{attribute 'GeneratedUsingTerminal: EK1100-0000-0018'}
{attribute addProperty BoxType "EK1100-0000-0018"}
{attribute addProperty Id "Beckhoff_EL72xxEK1122Beckhoff_EL72xxEK1122_48DD6FE82A_0001_EL7201_0000_0017EL7201_E258D19D33A_0002_EL7201_0000_0018EL7201_E258D19D33A_0003_EL7201_0000_0019EL7201_E258D19D33A_0004_EL7201_0000_0020EL7201_E258D19D33A_0005_EL7201_0000_0021EL7201_E258D19D33A_0006_EL7201_0001_0017EL7201_2B9C00AB33A_0007_EL7201_0001_0018EL7201_2B9C00AB33A_0008_EL7201_0001_0019EL7201_2B9C00AB33A_0009_EL7201_0001_0020EL7201_2B9C00AB33A_0010_EL7201_0001_0021EL7201_2B9C00AB33A_0011_EL7201_0010_0019EL7201_E258D19D33A_0012_EL7201_0010_0020EL7201_E258D19D33A_0013_EL7201_0010_0021EL7201_E258D19D33A_0014_EL7201_0010_0022EL7201_E258D19D33A_0015_EL7201_0010_0023EL7201_E258D19D33A_0016_EL7201_0010_0024EL7201_E258D19D33A_0017_EL7201_0010_0025EL7201_E258D19D33A_0018_EL7201_0010_0026EL7201_E258D19D33A_0019_EL7201_0010_0027EL7201_E258D19D33A_0020_EL7201_0010_0028EL7201_E258D19D33A_0021_EL7201_0010_0029EL7201_E258D19D33A_0022_EL7201_0010_0030EL7201_D07AE8BA34A_0023_EL7201_0010_0031EL7201_D07AE8BA34A_0024_EL7201_0010_0032EL7201_D07AE8BA34A_0025_EL7201_0011_0019EL7201_2B9C00AB33A_0026_EL7201_0011_0020EL7201_2B9C00AB33A_0027_EL7201_0011_0021EL7201_2B9C00AB33A_0028_EL7201_0011_0022EL7201_2B9C00AB33A_0029_EL7201_0011_0023EL7201_2B9C00AB33A_0030_EL7201_0011_0024EL7201_2B9C00AB33A_0031_EL7201_0011_0025EL7201_2B9C00AB33A_0032_EL7201_0011_0026EL7201_2B9C00AB33A_0033_EL7201_0011_0027EL7201_2B9C00AB33A_0034_EL7201_0011_0028EL7201_2B9C00AB33A_0035_EL7201_0011_0029EL7201_2B9C00AB33A_0036_EL7201_0011_0030EL7201_2B9C00AB33A_0037_EL7201_0011_0031EL7201_2B9C00AB33A_0038_EL7201_0011_0032EL7201_2B9C00AB33A_0039_EL7211_0000_0020EL7211_E258D19D33A_0040_EL7211_0000_0021EL7211_E258D19D33A_0041_EL7211_0001_0020EL7211_2B9C00AB33A_0042_EL7211_0001_0021EL7211_2B9C00AB33A_0043_EL7211_0010_0023EL7211_E258D19D33A_0044_EL7211_0010_0024EL7211_E258D19D33A_0045_EL7211_0010_0025EL7211_E258D19D33A_0046_EL7211_0010_0026EL7211_E258D19D33A_0047_EL7211_0010_0027EL7211_E258D19D33A_0048_EL7211_0010_0028EL7211_E258D19D33A_0049_EL7211_0010_0029EL7211_E258D19D33A_0050_EL7211_0010_0030EL7211_D07AE8BA34A_0051_EL7211_0010_0031EL7211_D07AE8BA34A_0052_EL7211_0010_0032EL7211_D07AE8BA34A_0053_EL7211_0011_0023EL7211_2B9C00AB33A_0054_EL7211_0011_0024EL7211_2B9C00AB33A_0055_EL7211_0011_0025EL7211_2B9C00AB33A_0056_EL7211_0011_0026EL7211_2B9C00AB33A_0057_EL7211_0011_0027EL7211_2B9C00AB33A_0058_EL7211_0011_0028EL7211_2B9C00AB33A_0059_EL7211_0011_0029EL7211_2B9C00AB33A_0060_EL7211_0011_0030EL7211_2B9C00AB33A_0061_EL7211_0011_0031EL7211_2B9C00AB33A_0062_EL7211_0011_0032EL7211_2B9C00AB33A_0063_EL7201_9014_0026EL7201_E258D19D33A_0064_EL7201_9014_0027EL7201_E258D19D33A_0065_EL7201_9014_0028EL7201_E258D19D33A_0066_EL7201_9014_0029EL7201_E258D19D33A_0067_EL7201_9014_0030EL7201_D07AE8BA34A_0068_EL7201_9014_0031EL7201_D07AE8BA34A_0069_EL7201_9014_0032EL7201_D07AE8BA34A_0070_EL7201_9015_0026EL7201_2B9C00AB33A_0071_EL7201_9015_0027EL7201_2B9C00AB33A_0072_EL7201_9015_0028EL7201_2B9C00AB33A_0073_EL7201_9015_0029EL7201_2B9C00AB33A_0074_EL7201_9015_0030EL7201_2B9C00AB33A_0075_EL7201_9015_0031EL7201_2B9C00AB33A_0076_EL7201_9015_0032EL7201_2B9C00AB33A_0077_EL7211_9014_0026EL7211_E258D19D33A_0078_EL7211_9014_0027EL7211_E258D19D33A_0079_EL7211_9014_0028EL7211_E258D19D33A_0080_EL7211_9014_0029EL7211_E258D19D33A_0081_EL7211_9014_0030EL7211_D07AE8BA34A_0082_EL7211_9014_0031EL7211_D07AE8BA34A_0083_EL7211_9014_0032EL7211_D07AE8BA34A_0084_EL7211_9015_0026EL7211_2B9C00AB33A_0085_EL7211_9015_0027EL7211_2B9C00AB33A_0086_EL7211_9015_0028EL7211_2B9C00AB33A_0087_EL7211_9015_0029EL7211_2B9C00AB33A_0088_EL7211_9015_0030EL7211_2B9C00AB33A_0089_EL7211_9015_0031EL7211_2B9C00AB33A_0090_EL7211_9015_0032EL7211_2B9C00AB33A_0091_EL7221_0000_0021EL7221_E258D19D33A_0092_EL7221_0001_0021EL7221_2B9C00AB33A_0093_EL7221_9014_0028EL7221_E258D19D33A_0094_EL7221_9014_0029EL7221_E258D19D33A_0095_EL7221_9014_0030EL7221_D07AE8BA34A_0096_EL7221_9014_0031EL7221_D07AE8BA34A_0097_EL7221_9014_0032EL7221_D07AE8BA34A_0098_EL7221_9015_0028EL7221_2B9C00AB33A_0099_EL7221_9015_0029EL7221_2B9C00AB33A_0100_EL7221_9015_0030EL7221_2B9C00AB33A_0101_EL7221_9015_0031EL7221_2B9C00AB33A_0102_EL7221_9015_0032EL7221_2B9C00AB33"}
{attribute addProperty CRC "2805504401"}
{attribute addProperty Size "3383"}
TYPE Beckhoff_EL72xx_A7389991 EXTENDS EK1100_AB5A9467 :
STRUCT
	{attribute addProperty Name "Beckhoff_EL72xxEK1122"}
	Beckhoff_EL72xxEK1122 : Beckhoff_EL72xxEK1122_48DD6FE8;
	{attribute addProperty Name "A_0001_EL7201_0000_0017"}
	A_0001_EL7201_0000_0017 : EL7201_E258D19D;
	{attribute addProperty Name "A_0002_EL7201_0000_0018"}
	A_0002_EL7201_0000_0018 : EL7201_E258D19D;
	{attribute addProperty Name "A_0003_EL7201_0000_0019"}
	A_0003_EL7201_0000_0019 : EL7201_E258D19D;
	{attribute addProperty Name "A_0004_EL7201_0000_0020"}
	A_0004_EL7201_0000_0020 : EL7201_E258D19D;
	{attribute addProperty Name "A_0005_EL7201_0000_0021"}
	A_0005_EL7201_0000_0021 : EL7201_E258D19D;
	{attribute addProperty Name "A_0006_EL7201_0001_0017"}
	A_0006_EL7201_0001_0017 : EL7201_2B9C00AB;
	{attribute addProperty Name "A_0007_EL7201_0001_0018"}
	A_0007_EL7201_0001_0018 : EL7201_2B9C00AB;
	{attribute addProperty Name "A_0008_EL7201_0001_0019"}
	A_0008_EL7201_0001_0019 : EL7201_2B9C00AB;
	{attribute addProperty Name "A_0009_EL7201_0001_0020"}
	A_0009_EL7201_0001_0020 : EL7201_2B9C00AB;
	{attribute addProperty Name "A_0010_EL7201_0001_0021"}
	A_0010_EL7201_0001_0021 : EL7201_2B9C00AB;
	{attribute addProperty Name "A_0011_EL7201_0010_0019"}
	A_0011_EL7201_0010_0019 : EL7201_E258D19D;
	{attribute addProperty Name "A_0012_EL7201_0010_0020"}
	A_0012_EL7201_0010_0020 : EL7201_E258D19D;
	{attribute addProperty Name "A_0013_EL7201_0010_0021"}
	A_0013_EL7201_0010_0021 : EL7201_E258D19D;
	{attribute addProperty Name "A_0014_EL7201_0010_0022"}
	A_0014_EL7201_0010_0022 : EL7201_E258D19D;
	{attribute addProperty Name "A_0015_EL7201_0010_0023"}
	A_0015_EL7201_0010_0023 : EL7201_E258D19D;
	{attribute addProperty Name "A_0016_EL7201_0010_0024"}
	A_0016_EL7201_0010_0024 : EL7201_E258D19D;
	{attribute addProperty Name "A_0017_EL7201_0010_0025"}
	A_0017_EL7201_0010_0025 : EL7201_E258D19D;
	{attribute addProperty Name "A_0018_EL7201_0010_0026"}
	A_0018_EL7201_0010_0026 : EL7201_E258D19D;
	{attribute addProperty Name "A_0019_EL7201_0010_0027"}
	A_0019_EL7201_0010_0027 : EL7201_E258D19D;
	{attribute addProperty Name "A_0020_EL7201_0010_0028"}
	A_0020_EL7201_0010_0028 : EL7201_E258D19D;
	{attribute addProperty Name "A_0021_EL7201_0010_0029"}
	A_0021_EL7201_0010_0029 : EL7201_E258D19D;
	{attribute addProperty Name "A_0022_EL7201_0010_0030"}
	A_0022_EL7201_0010_0030 : EL7201_D07AE8BA;
	{attribute addProperty Name "A_0023_EL7201_0010_0031"}
	A_0023_EL7201_0010_0031 : EL7201_D07AE8BA;
	{attribute addProperty Name "A_0024_EL7201_0010_0032"}
	A_0024_EL7201_0010_0032 : EL7201_D07AE8BA;
	{attribute addProperty Name "A_0025_EL7201_0011_0019"}
	A_0025_EL7201_0011_0019 : EL7201_2B9C00AB;
	{attribute addProperty Name "A_0026_EL7201_0011_0020"}
	A_0026_EL7201_0011_0020 : EL7201_2B9C00AB;
	{attribute addProperty Name "A_0027_EL7201_0011_0021"}
	A_0027_EL7201_0011_0021 : EL7201_2B9C00AB;
	{attribute addProperty Name "A_0028_EL7201_0011_0022"}
	A_0028_EL7201_0011_0022 : EL7201_2B9C00AB;
	{attribute addProperty Name "A_0029_EL7201_0011_0023"}
	A_0029_EL7201_0011_0023 : EL7201_2B9C00AB;
	{attribute addProperty Name "A_0030_EL7201_0011_0024"}
	A_0030_EL7201_0011_0024 : EL7201_2B9C00AB;
	{attribute addProperty Name "A_0031_EL7201_0011_0025"}
	A_0031_EL7201_0011_0025 : EL7201_2B9C00AB;
	{attribute addProperty Name "A_0032_EL7201_0011_0026"}
	A_0032_EL7201_0011_0026 : EL7201_2B9C00AB;
	{attribute addProperty Name "A_0033_EL7201_0011_0027"}
	A_0033_EL7201_0011_0027 : EL7201_2B9C00AB;
	{attribute addProperty Name "A_0034_EL7201_0011_0028"}
	A_0034_EL7201_0011_0028 : EL7201_2B9C00AB;
	{attribute addProperty Name "A_0035_EL7201_0011_0029"}
	A_0035_EL7201_0011_0029 : EL7201_2B9C00AB;
	{attribute addProperty Name "A_0036_EL7201_0011_0030"}
	A_0036_EL7201_0011_0030 : EL7201_2B9C00AB;
	{attribute addProperty Name "A_0037_EL7201_0011_0031"}
	A_0037_EL7201_0011_0031 : EL7201_2B9C00AB;
	{attribute addProperty Name "A_0038_EL7201_0011_0032"}
	A_0038_EL7201_0011_0032 : EL7201_2B9C00AB;
	{attribute addProperty Name "A_0039_EL7211_0000_0020"}
	A_0039_EL7211_0000_0020 : EL7211_E258D19D;
	{attribute addProperty Name "A_0040_EL7211_0000_0021"}
	A_0040_EL7211_0000_0021 : EL7211_E258D19D;
	{attribute addProperty Name "A_0041_EL7211_0001_0020"}
	A_0041_EL7211_0001_0020 : EL7211_2B9C00AB;
	{attribute addProperty Name "A_0042_EL7211_0001_0021"}
	A_0042_EL7211_0001_0021 : EL7211_2B9C00AB;
	{attribute addProperty Name "A_0043_EL7211_0010_0023"}
	A_0043_EL7211_0010_0023 : EL7211_E258D19D;
	{attribute addProperty Name "A_0044_EL7211_0010_0024"}
	A_0044_EL7211_0010_0024 : EL7211_E258D19D;
	{attribute addProperty Name "A_0045_EL7211_0010_0025"}
	A_0045_EL7211_0010_0025 : EL7211_E258D19D;
	{attribute addProperty Name "A_0046_EL7211_0010_0026"}
	A_0046_EL7211_0010_0026 : EL7211_E258D19D;
	{attribute addProperty Name "A_0047_EL7211_0010_0027"}
	A_0047_EL7211_0010_0027 : EL7211_E258D19D;
	{attribute addProperty Name "A_0048_EL7211_0010_0028"}
	A_0048_EL7211_0010_0028 : EL7211_E258D19D;
	{attribute addProperty Name "A_0049_EL7211_0010_0029"}
	A_0049_EL7211_0010_0029 : EL7211_E258D19D;
	{attribute addProperty Name "A_0050_EL7211_0010_0030"}
	A_0050_EL7211_0010_0030 : EL7211_D07AE8BA;
	{attribute addProperty Name "A_0051_EL7211_0010_0031"}
	A_0051_EL7211_0010_0031 : EL7211_D07AE8BA;
	{attribute addProperty Name "A_0052_EL7211_0010_0032"}
	A_0052_EL7211_0010_0032 : EL7211_D07AE8BA;
	{attribute addProperty Name "A_0053_EL7211_0011_0023"}
	A_0053_EL7211_0011_0023 : EL7211_2B9C00AB;
	{attribute addProperty Name "A_0054_EL7211_0011_0024"}
	A_0054_EL7211_0011_0024 : EL7211_2B9C00AB;
	{attribute addProperty Name "A_0055_EL7211_0011_0025"}
	A_0055_EL7211_0011_0025 : EL7211_2B9C00AB;
	{attribute addProperty Name "A_0056_EL7211_0011_0026"}
	A_0056_EL7211_0011_0026 : EL7211_2B9C00AB;
	{attribute addProperty Name "A_0057_EL7211_0011_0027"}
	A_0057_EL7211_0011_0027 : EL7211_2B9C00AB;
	{attribute addProperty Name "A_0058_EL7211_0011_0028"}
	A_0058_EL7211_0011_0028 : EL7211_2B9C00AB;
	{attribute addProperty Name "A_0059_EL7211_0011_0029"}
	A_0059_EL7211_0011_0029 : EL7211_2B9C00AB;
	{attribute addProperty Name "A_0060_EL7211_0011_0030"}
	A_0060_EL7211_0011_0030 : EL7211_2B9C00AB;
	{attribute addProperty Name "A_0061_EL7211_0011_0031"}
	A_0061_EL7211_0011_0031 : EL7211_2B9C00AB;
	{attribute addProperty Name "A_0062_EL7211_0011_0032"}
	A_0062_EL7211_0011_0032 : EL7211_2B9C00AB;
	{attribute addProperty Name "A_0063_EL7201_9014_0026"}
	A_0063_EL7201_9014_0026 : EL7201_E258D19D;
	{attribute addProperty Name "A_0064_EL7201_9014_0027"}
	A_0064_EL7201_9014_0027 : EL7201_E258D19D;
	{attribute addProperty Name "A_0065_EL7201_9014_0028"}
	A_0065_EL7201_9014_0028 : EL7201_E258D19D;
	{attribute addProperty Name "A_0066_EL7201_9014_0029"}
	A_0066_EL7201_9014_0029 : EL7201_E258D19D;
	{attribute addProperty Name "A_0067_EL7201_9014_0030"}
	A_0067_EL7201_9014_0030 : EL7201_D07AE8BA;
	{attribute addProperty Name "A_0068_EL7201_9014_0031"}
	A_0068_EL7201_9014_0031 : EL7201_D07AE8BA;
	{attribute addProperty Name "A_0069_EL7201_9014_0032"}
	A_0069_EL7201_9014_0032 : EL7201_D07AE8BA;
	{attribute addProperty Name "A_0070_EL7201_9015_0026"}
	A_0070_EL7201_9015_0026 : EL7201_2B9C00AB;
	{attribute addProperty Name "A_0071_EL7201_9015_0027"}
	A_0071_EL7201_9015_0027 : EL7201_2B9C00AB;
	{attribute addProperty Name "A_0072_EL7201_9015_0028"}
	A_0072_EL7201_9015_0028 : EL7201_2B9C00AB;
	{attribute addProperty Name "A_0073_EL7201_9015_0029"}
	A_0073_EL7201_9015_0029 : EL7201_2B9C00AB;
	{attribute addProperty Name "A_0074_EL7201_9015_0030"}
	A_0074_EL7201_9015_0030 : EL7201_2B9C00AB;
	{attribute addProperty Name "A_0075_EL7201_9015_0031"}
	A_0075_EL7201_9015_0031 : EL7201_2B9C00AB;
	{attribute addProperty Name "A_0076_EL7201_9015_0032"}
	A_0076_EL7201_9015_0032 : EL7201_2B9C00AB;
	{attribute addProperty Name "A_0077_EL7211_9014_0026"}
	A_0077_EL7211_9014_0026 : EL7211_E258D19D;
	{attribute addProperty Name "A_0078_EL7211_9014_0027"}
	A_0078_EL7211_9014_0027 : EL7211_E258D19D;
	{attribute addProperty Name "A_0079_EL7211_9014_0028"}
	A_0079_EL7211_9014_0028 : EL7211_E258D19D;
	{attribute addProperty Name "A_0080_EL7211_9014_0029"}
	A_0080_EL7211_9014_0029 : EL7211_E258D19D;
	{attribute addProperty Name "A_0081_EL7211_9014_0030"}
	A_0081_EL7211_9014_0030 : EL7211_D07AE8BA;
	{attribute addProperty Name "A_0082_EL7211_9014_0031"}
	A_0082_EL7211_9014_0031 : EL7211_D07AE8BA;
	{attribute addProperty Name "A_0083_EL7211_9014_0032"}
	A_0083_EL7211_9014_0032 : EL7211_D07AE8BA;
	{attribute addProperty Name "A_0084_EL7211_9015_0026"}
	A_0084_EL7211_9015_0026 : EL7211_2B9C00AB;
	{attribute addProperty Name "A_0085_EL7211_9015_0027"}
	A_0085_EL7211_9015_0027 : EL7211_2B9C00AB;
	{attribute addProperty Name "A_0086_EL7211_9015_0028"}
	A_0086_EL7211_9015_0028 : EL7211_2B9C00AB;
	{attribute addProperty Name "A_0087_EL7211_9015_0029"}
	A_0087_EL7211_9015_0029 : EL7211_2B9C00AB;
	{attribute addProperty Name "A_0088_EL7211_9015_0030"}
	A_0088_EL7211_9015_0030 : EL7211_2B9C00AB;
	{attribute addProperty Name "A_0089_EL7211_9015_0031"}
	A_0089_EL7211_9015_0031 : EL7211_2B9C00AB;
	{attribute addProperty Name "A_0090_EL7211_9015_0032"}
	A_0090_EL7211_9015_0032 : EL7211_2B9C00AB;
	{attribute addProperty Name "A_0091_EL7221_0000_0021"}
	A_0091_EL7221_0000_0021 : EL7221_E258D19D;
	{attribute addProperty Name "A_0092_EL7221_0001_0021"}
	A_0092_EL7221_0001_0021 : EL7221_2B9C00AB;
	{attribute addProperty Name "A_0093_EL7221_9014_0028"}
	A_0093_EL7221_9014_0028 : EL7221_E258D19D;
	{attribute addProperty Name "A_0094_EL7221_9014_0029"}
	A_0094_EL7221_9014_0029 : EL7221_E258D19D;
	{attribute addProperty Name "A_0095_EL7221_9014_0030"}
	A_0095_EL7221_9014_0030 : EL7221_D07AE8BA;
	{attribute addProperty Name "A_0096_EL7221_9014_0031"}
	A_0096_EL7221_9014_0031 : EL7221_D07AE8BA;
	{attribute addProperty Name "A_0097_EL7221_9014_0032"}
	A_0097_EL7221_9014_0032 : EL7221_D07AE8BA;
	{attribute addProperty Name "A_0098_EL7221_9015_0028"}
	A_0098_EL7221_9015_0028 : EL7221_2B9C00AB;
	{attribute addProperty Name "A_0099_EL7221_9015_0029"}
	A_0099_EL7221_9015_0029 : EL7221_2B9C00AB;
	{attribute addProperty Name "A_0100_EL7221_9015_0030"}
	A_0100_EL7221_9015_0030 : EL7221_2B9C00AB;
	{attribute addProperty Name "A_0101_EL7221_9015_0031"}
	A_0101_EL7221_9015_0031 : EL7221_2B9C00AB;
	{attribute addProperty Name "A_0102_EL7221_9015_0032"}
	A_0102_EL7221_9015_0032 : EL7221_2B9C00AB;
END_STRUCT
END_TYPE

(* stored: Version 1.2.0.0, ProductVersion 3.1.4024.9
   DUT Beckhoff_EL72xx_A7389991: Id {a740abac-b79f-4667-8675-ca733c229be8} *)
